// TIA Portal V20 export
FUNCTION_BLOCK "SysBaluffBUS007F"   // FB4010, FBD
{ S7_Optimized_Access := 'TRUE' }
// stored: AutoNumber false, MemoryReserve 100, SetENOAutomatically false
   VAR_INPUT
      adrHW { ExternalAccessible := 'False'; ExternalVisible := 'False'; ExternalWritable := 'False'} : HW_IO;   // I/O adress HW / I/O adress
      adr { ExternalAccessible := 'False'; ExternalVisible := 'False'; ExternalWritable := 'False'} : Int;   // I/O adress
      slot { ExternalAccessible := 'False'; ExternalVisible := 'False'; ExternalWritable := 'False'} : Int;   // slot of io link module 1..4
      ack { ExternalAccessible := 'False'; ExternalVisible := 'False'; ExternalWritable := 'False'} : Bool;   // acknowledge
      startConfig { ExternalAccessible := 'False'; ExternalVisible := 'False'; ExternalWritable := 'False'} : Bool;
   END_VAR
   VAR_OUTPUT
      Measure { ExternalAccessible := 'False'; ExternalVisible := 'False'; ExternalWritable := 'False'} : Real;   // Actual measured value [mm] (-1= Read error)
      Scale { ExternalAccessible := 'False'; ExternalVisible := 'False'; ExternalWritable := 'False'} : Real;   // Scale -1 = 1/10mm
      ComOk { ExternalAccessible := 'False'; ExternalVisible := 'False'; ExternalWritable := 'False'} : Bool;   // communication ok
      ConfigOk { ExternalAccessible := 'False'; ExternalVisible := 'False'; ExternalWritable := 'False'} : Bool;   // configuration ok
      MeasureOk { ExternalAccessible := 'False'; ExternalVisible := 'False'; ExternalWritable := 'False'} : Bool;   // measuring ok
      Err { ExternalAccessible := 'False'; ExternalVisible := 'False'; ExternalWritable := 'False'} : Bool;   // Signal sensor error (1= Error)
      Warn { ExternalAccessible := 'False'; ExternalVisible := 'False'; ExternalWritable := 'False'} : Bool;   // Signal sensorwarning (1= Dirty)
      A1 { ExternalAccessible := 'False'; ExternalVisible := 'False'; ExternalWritable := 'False'} : Bool;   // Signal output 1 (1= Occ)
   END_VAR
   VAR_IN_OUT
      param : "TypeIOLinkParamArray";
   END_VAR
   VAR
      var { ExternalAccessible := 'False'; ExternalVisible := 'False'; ExternalWritable := 'False'} : Struct
         "bool" : Bool;
         "byte" : Byte;
         "word" : Word;
         "dword" : DWord;
         "int" : Int;
         "dint" : DInt;
         "real" : Real;
         s5time : S5Time;
         "time" : Time;
         hm : Array[1..50] of Bool;
         fm : Array[1..50] of Bool;
      END_STRUCT;
      Rd { ExternalAccessible := 'False'; ExternalVisible := 'False'; ExternalWritable := 'False'} : "TypeBaluffBUS007xRd";
      Data { ExternalAccessible := 'False'; ExternalVisible := 'False'; ExternalWritable := 'False'} : Struct
         Measure : Real;
         Scale : Real;
         ComOk : Bool;
         ConfigOk : Bool;
         MeasureOk : Bool;
         A1 : Bool;
         A2 : Bool;
         Warn : Bool;
         Err : Bool;
         ErrCom : Bool;
         ErrSensor : Bool;
         ErrConfig : Bool;
         WarnSensor : Bool;
      END_STRUCT;
      device { ExternalAccessible := 'False'; ExternalVisible := 'False'; ExternalWritable := 'False'} : "LIOLink_Device";
      statRecord { ExternalAccessible := 'False'; ExternalVisible := 'False'; ExternalWritable := 'False'} : Array[0..231] of Byte;
      cfgData { ExternalAccessible := 'False'; ExternalVisible := 'False'; ExternalWritable := 'False'} : Struct
         Index : Int;
         Subindex : Int;
         Len : Int;
         Value : "TypeIOLinkParamData";
      END_STRUCT;
      cfg { ExternalAccessible := 'False'; ExternalVisible := 'False'; ExternalWritable := 'False'} : Struct
         "Step" : Int;
         Done : Bool;
         Active : Bool;
         Err : Bool;
         Restart : Bool;
      END_STRUCT;
      T1 { ExternalAccessible := 'False'; ExternalVisible := 'False'; ExternalWritable := 'False'} : TON_TIME;
      cnt_i { ExternalAccessible := 'False'; ExternalVisible := 'False'; ExternalWritable := 'False'} : Int;
      cnt_y { ExternalAccessible := 'False'; ExternalVisible := 'False'; ExternalWritable := 'False'} : Int;
      cnt_x { ExternalAccessible := 'False'; ExternalVisible := 'False'; ExternalWritable := 'False'} : Int;
   END_VAR
   VAR_TEMP
      t_Data1 : Word;
      t_Data2 : Byte;
      t_Data3 : Byte;
      t_ENO : Bool;
   END_VAR
BEGIN

REGION Network 1 (SCL): info
   (*            
       Serie:          Baluff BUS007F  
       Type:           Baluff BUS M18M1-GPXI-03/025-S92G-511
       Range:          30..350mm
       Vendor ID:      888
       Device ID:      264209
       Input:          4 Byte
       Output:         0 Byte   

       Autor:          Alexander Kiebacher
       Datum:          05/2024
       Änderung:       05/2024
       Version:        1.0
       Lizenz:         Microtec

       Revisionen:     V1.0
   *)
END_REGION

REGION Network 2 (SCL): read data

   #t_Data1 := PEEK_WORD(area := 16#1, dbNumber := 0, byteOffset := #adr, ENO => #t_ENO);
   #t_Data2 := PEEK_BYTE(area := 16#1, dbNumber := 0, byteOffset := #adr + 2, ENO => #t_ENO);
   #t_Data3 := PEEK_BYTE(area := 16#1, dbNumber := 0, byteOffset := #adr + 3, ENO => #t_ENO);
   ENO := #t_ENO;
END_REGION

REGION Network 3 (SCL): read data - copy data
   // #Data.Scale := WORD_TO_SINT(SHR(IN := #t_Data2 AND 16#FF00, N := 8));
   // 
   // 0x80000008 –2147483640 Objekt zu nah
   // 0x7FFFFFF8 2147483640 Objekt zu weit
   // 0x7FFFFFFC 2147483644 Kein Signal

   IF ENO THEN

       #Rd.Measure := WORD_TO_INT(#t_Data1);
       #Rd.Scale := BYTE_TO_SINT(#t_Data2);

       #Rd.SCC1 := #t_Data3.%X0;

       // check communication
       #Data.MeasureOk := false;
       IF #Rd.Measure <> 0 THEN
           #Data.ComOk := true;
       ELSE
           #Data.ComOk := false;
       END_IF;

       IF #Rd.Measure = 32764 THEN             // no measurement data
           #Data.Measure := -1.0;
       ELSIF #Rd.Measure <= -32760 THEN        // out of measuring range (-)
           #Data.Measure := -1.0;
       ELSIF #Rd.Measure >= 32760 THEN         // out of measuring range (+)
           #Data.Measure := -1.0;
       ELSIF #Data.ComOk THEN
           #Data.Measure := INT_TO_REAL(#Rd.Measure) / 10.0;
           #Data.MeasureOk := true;
       END_IF;


       #Data.Scale := SINT_TO_REAL(#Rd.Scale);
       #Data.A1 := #Rd.SCC1;
       #Data.A2 := false;

   ELSE
       #Data.Measure := -1.0;
       #Data.Scale := 0.0;
       #Data.A1 := false;
       #Data.A2 := false;
       #Data.ComOk := false;

   END_IF;
END_REGION

REGION Network 5: reset fault / warning / reset faults
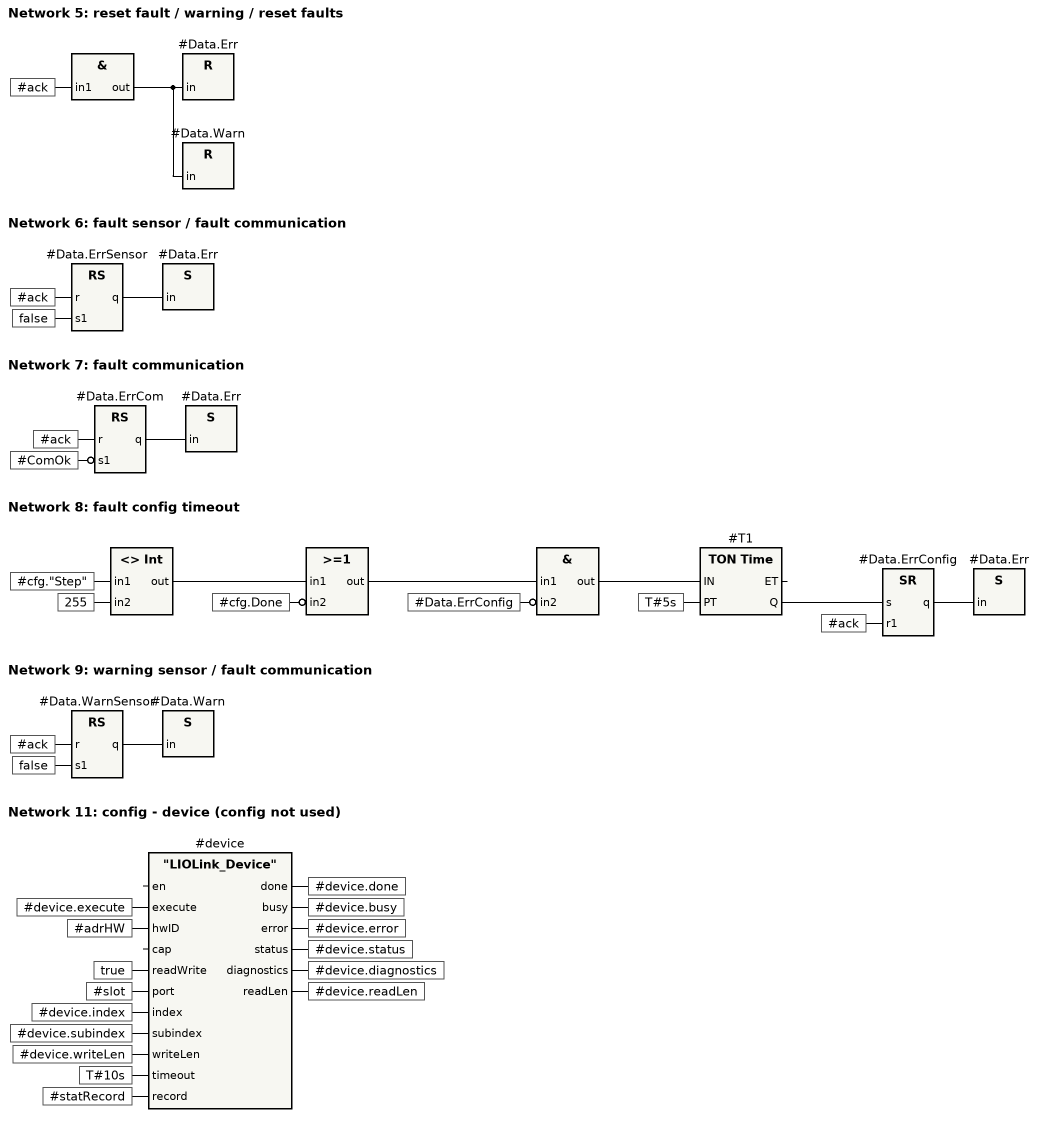
   IF #ack THEN
       #Data.Err := FALSE;
       #Data.Warn := FALSE;
   END_IF;
END_REGION

REGION Network 6: fault sensor / fault communication
   IF #ack THEN
       #Data.ErrSensor := FALSE;   // RS flip-flop
   END_IF;
   IF false THEN #Data.ErrSensor := TRUE; END_IF;
   IF #Data.ErrSensor THEN #Data.Err := TRUE; END_IF;
END_REGION

REGION Network 7: fault communication
   IF #ack THEN
       #Data.ErrCom := FALSE;   // RS flip-flop
   END_IF;
   IF NOT #ComOk THEN #Data.ErrCom := TRUE; END_IF;
   IF #Data.ErrCom THEN #Data.Err := TRUE; END_IF;
END_REGION

REGION Network 8: fault config timeout
   #T1(IN := ((#cfg."Step" <> 255) OR NOT #cfg.Done) AND NOT #Data.ErrConfig, PT := T#5s);   // TON
   IF #T1.Q THEN
       #Data.ErrConfig := TRUE;   // SR flip-flop
   END_IF;
   IF #ack THEN #Data.ErrConfig := FALSE; END_IF;
   IF #Data.ErrConfig THEN #Data.Err := TRUE; END_IF;
END_REGION

REGION Network 9: warning sensor / fault communication
   IF #ack THEN
       #Data.WarnSensor := FALSE;   // RS flip-flop
   END_IF;
   IF false THEN #Data.WarnSensor := TRUE; END_IF;
   IF #Data.WarnSensor THEN #Data.Warn := TRUE; END_IF;
END_REGION

REGION Network 11: config - device (config not used)
   #device(execute := #device.execute,   // "LIOLink_Device"
           hwID := #adrHW,
           readWrite := true,
           port := #slot,
           index := #device.index,
           subindex := #device.subindex,
           writeLen := #device.writeLen,
           timeout := T#10s,
           record := #statRecord,
           done => #device.done,
           busy => #device.busy,
           error => #device.error,
           status => #device.status,
           diagnostics => #device.diagnostics,
           readLen => #device.readLen);
END_REGION

REGION Network 12 (SCL): config - device (config not used)
   (* Invalid *)

   IF (#cfg.Step <= 0 OR #cfg.Step > 255 OR #Data.ErrConfig) THEN
       #cfg.Done := false;
       #cfg.Err := true;
       #cfg.Step := 1;
       #device.execute := false;
   END_IF;

   CASE #cfg.Step OF
       1:  (* Not configured or config request *)
           IF (NOT #cfg.Done OR #cfg.Restart) AND NOT #Data.ErrConfig THEN
               #cfg.Done := false;
               #cfg.Restart := false;
               #cfg.Err := true;
               #cfg.Step := 20;
               #cnt_i := 0;
               #device.execute := false;
           END_IF;

   (* Setup correct operation mode *)        
       20: (* Start config  *)

           #cfgData.Index := #param.Param[#cnt_i].Index;
           #cfgData.Subindex := #param.Param[#cnt_i].Subindex;
           #cfgData.Len := #param.Param[#cnt_i].Len;

           FOR #cnt_y := 0 TO (#cfgData.Len - 1) BY 1 DO
               #cfgData.Value.data[#cnt_y] := #param.Param[#cnt_i].Value.data[#cnt_y];
           END_FOR;

           #device.index := #cfgData.Index ;
           #device.subindex := #cfgData.Subindex ;
           #device.writeLen := #cfgData.Len;
           FOR #cnt_x := 0 TO (#cfgData.Len - 1) BY 1 DO
               #statRecord[#cnt_x] := #cfgData.Value.data[#cnt_x];
           END_FOR;

           #device.execute := false;
           #cfg.Step := 21;

       21: (* Start request *)
           #device.execute := true;
           #cfg.Step := 22;

       22: (*Wait for execution *)
           IF #device.done THEN
               #device.execute := false;
               IF #param.Param[#cnt_i + 1].Len <> 0 THEN
                   #cnt_i := #cnt_i + 1;
                   #cfg.Step := 20;
               ELSE
                   #cfg.Step := 255;
               END_IF;

           END_IF;
           IF #device.error THEN
               #device.execute := false;
               #cfg.Step := 20;
           END_IF;

   (* Setup done *)
       255:
           #cfg.Done := true;
           #cfg.Err := false;

           IF #cfg.Done AND #startConfig THEN
               #cfg.Done := false;
               #cfg.Err := true;
               #cfg.Step := 1;
               #device.execute := false;
               #Data.ErrConfig := false;
           END_IF;

   END_CASE;

   #cfg.Active := #cfg.Step > 10 AND #cfg.Step <255;

   #Data.ConfigOk := #cfg.Done;

   IF TRUE THEN

       #Data.ConfigOk := TRUE;
       #cfg.Done := TRUE;
       #cfg.Step := 255;

   END_IF;
END_REGION

REGION Network 13 (SCL): write outputs

   #Measure := #Data.Measure;
   #Scale := #Data.Scale;
   #ComOk := #Data.ComOk;
   #ConfigOk := #Data.ConfigOk;
   #MeasureOk := #Data.MeasureOk;
   #Err := #Data.Err;
   #Warn := #Data.Warn;
   #A1 := #Data.A1;
END_REGION
END_FUNCTION_BLOCK
